// TIA Portal V19 export
TYPE "LAF_typeReferenceConfiguration"
// stored: Access Published
   STRUCT
      parent : WString[128];   // Reference designator for describing the parent module
      relative : WString[25] := WSTRING#'';   // Reference designator for describing the own module
      combined : WString[128];   // Do not change. Will be created automatically
   END_STRUCT;
END_TYPE
